(* Logix 5000 project; controller cal1615 1756-L62 rev 16.20; software revision 16.05; part 23 of 78 *)
(* tags used below, declared in another part *)
   FAULT : BOOL;   // Fault AFI
   HMI : BOOL;   // AFI HMI
   p01r09_pb_global_reset : BOOL;   // System Modes PB: Global Fault Reset
   p12_ai_exhaust_amps : REAL;   // Zone 2 Analog Input Exhaust Fan Amps
   p12_ai_exhaust_hz : REAL;   // Zone 2 Analog Input Exhaust Fan HZ
   p12_ai_exhaust_pct : REAL;   // Zone 2 Analog Input Exhaust Fan PCT
   p12_ai_exhaust_rpm : REAL;   // Zone 2 Analog Input Exhaust Fan RPM
   p12_ai_lfl : REAL;   // Zone 2 Analog Input Lower Flash Limit
   p12_ai_prs : REAL;   // Zone 2 Analog Input Pressure
   p12_ai_recirc_amps : REAL;   // Zone 2 Analog Input Recirc Fan Amps
   p12_ai_recirc_hz : REAL;   // Zone 2 Analog Input Supply Fan HZ
   p12_ai_recirc_pct : REAL;   // Zone 2 Analog Input Recirc Fan PCT
   p12_ai_recirc_rpm : REAL;   // Zone 2 Analog Input Recirc Fan RPM
   p12_ai_tc01 : REAL;   // Zone 2 Analog Input Control Thermocouple 1
   p12_ai_tc02 : REAL;   // Zone 2 Analog Input Control Thermocouple 2
   p12_ao_cv : REAL;   // Zone 2 Analog Output Control Valve
   p12_ao_exhaust_selected_speed : REAL;   // Zone 2 Analog Output Exhaust Fan VFD Selected Speed
   p12_ao_recirc_selected_speed : REAL;   // Zone 2 Analog Output Recirc Fan VFD Selected Speed
   p12_di_burner_auto : BOOL;   // Zone 2 Digital Input Burner Auto
   p12_di_exh : acs800_di_normal;   // Zone 2 Digital Inputs Exhaust Fan
   p12_di_recirc : acs800_di_normal;   // Zone 2 Digital Inputs Recirc Fan
   p12_dint_to_hmi : DINT[16];   // Zone 2 Temperature Control VFDs On
   p12_param_fast_to_soak : REAL;   // Zone 2 Parameter Fast to Soak Control
   p12_param_lfl_hhl : REAL;   // Zone 2 Parameter High High Lower Flash Limit
   p12_param_lfl_hl : REAL;   // Zone 2 Parameter High LFL Limit
   p12_param_pid1_ff : REAL;   // Zone 2 Parameter Fast PID Bias
   p12_param_pid1_kd : REAL;   // Zone 2 Parameter Fast PID Derivative Gain
   p12_param_pid1_ki : REAL;   // Zone 2 Parameter Fast PID Integral Gain
   p12_param_pid1_kp : REAL;   // Zone 2 Parameter Fast PID Proportional Gain
   p12_param_pid2_ff : REAL;   // Zone 2 Parameter Auto PID Bias
   p12_param_pid2_kd : REAL;   // Zone 2 Parameter Auto PID Derivative Gain
   p12_param_pid2_ki : REAL;   // Zone 2 Parameter Auto PID Integral Gain
   p12_param_pid2_kp : REAL;   // Zone 2 Parameter Auto PID Proportional Gain
   p12_param_shutdown_temp : REAL;   // Zone 2 Parameter Zone Shutdown Temperature
   p12_param_soak_to_fast : REAL;   // Zone 2 Parameter Soak to Fast Control
   p12_param_tc01_dev : REAL;   // Zone 2 Parameter Oven Temperature Deviation from Setpoint
   p12_param_tc01_hl : REAL;   // Zone 2 Parameter Process Air High Limit
   p12_param_tc01z : REAL;   // Zone 2 Parameter Process Temperature Zero Offset
   p12_param_tc02z : REAL;   // Zone 2 Parameter SupplyTemperature Zero Offset
   p12_param_zone_pressure : REAL;   // Zone 2 Parameter High Pressure LImit
   p12_real_to_hmi : REAL[112];   // Zone 2 Real to HMI
   p12r01 : routine;   // Zone 2 Main
   p12r05 : routine;   // Zone 2 Dint to HMI
   p12r05_exh_status : DINT;
   p12r05_recirc_status : DINT;
   p12r05_Temp_ctl_status : DINT;
   p12r05_timer_fault : TIMER[4];   // Zone 2 Dint to HMI Fault Delay
   p12r05_timer_warning : TIMER[4];   // Zone 2 Dint to HMI Warning Delay
   p12r06 : routine;   // Zone 2 Real to HMI
   p12r06_timer_fault : TIMER[4];   // Zone 2 Real to HMI Fault Delay
   p12r06_timer_warning : TIMER[4];   // Zone 2 Real to HMI Warning Delay
   p12r07 : routine;   // Zone 2 Alarms
   p12r07_timer_fault : TIMER[4];   // Zone 2 Alarms Fault Delay
   p12r07_timer_warning : TIMER[4];   // Zone 2 Alarms Warning Delay
   p12r20 : routine;   // Zone 2 Temp Sequence
   p12r20_state : DINT;   // Zone 2 Temperature Control State
   p12r20_status : DINT;   // Zone 2 Temperature Control Sequence Status
   p12r30 : routine;   // Zone 2 Temperature Control
   p12r30_cv_man_sp : REAL;   // Zone 2 Temperature Control Manual Heat Control Valve Setpoint
   p12r30_permissive_run : BOOL;   // Zone 2 Temperature Control Run Permissive
   p12r30_pid_temp : PID;   // Zone 2 Temperature Control PID
   p12r30_pid_temp_pv : REAL;   // Zone 2 Temperature Control PID Temp Process Variable
   p12r30_pid_temp_sp : REAL;   // Zone 2 Temperature Control PID Temperature Control Setpoint
   p12r30_request_heat : BOOL;   // Zone 2 Temperature Control Request Heat
   p12r31 : routine;   // Zone 2 Exhaust VFD
   p12r31_vfd_stopped : BOOL;   // Zone 2 Exhaust VFD VFD Stopped
   p12r32 : routine;   // Zone 2 Recirc VFD
   p12r32_vfd_stopped : BOOL;   // Zone 2 Recirc VFD VFD Stopped
(* P12_Zone_2, continued *)

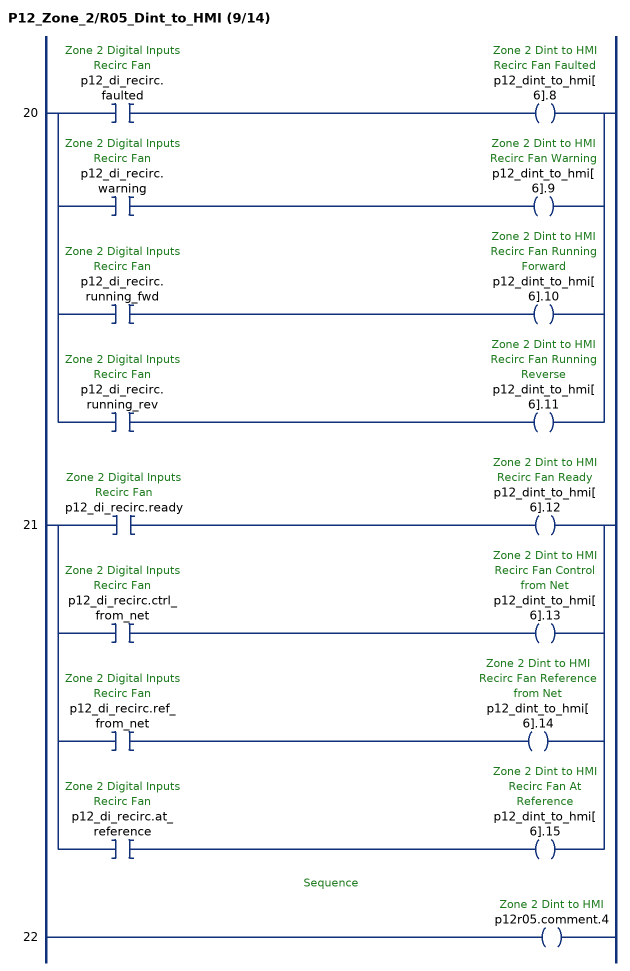
   [picture p388: P12_Zone_2/R05_Dint_to_HMI rungs 20-22]
   20: [XIC(p12_di_recirc.faulted) OTE(p12_dint_to_hmi[6].8) ,XIC(p12_di_recirc.warning) OTE(p12_dint_to_hmi[6].9) ,XIC(p12_di_recirc.running_fwd) OTE(p12_dint_to_hmi[6].10) ,XIC(p12_di_recirc.running_rev) OTE(p12_dint_to_hmi[6].11) ];
   21: [XIC(p12_di_recirc.ready) OTE(p12_dint_to_hmi[6].12) ,XIC(p12_di_recirc.ctrl_from_net) OTE(p12_dint_to_hmi[6].13) ,XIC(p12_di_recirc.ref_from_net) OTE(p12_dint_to_hmi[6].14) ,XIC(p12_di_recirc.at_reference) OTE(p12_dint_to_hmi[6].15) ];
   // Sequence
   22: OTE(p12r05.comment.4);
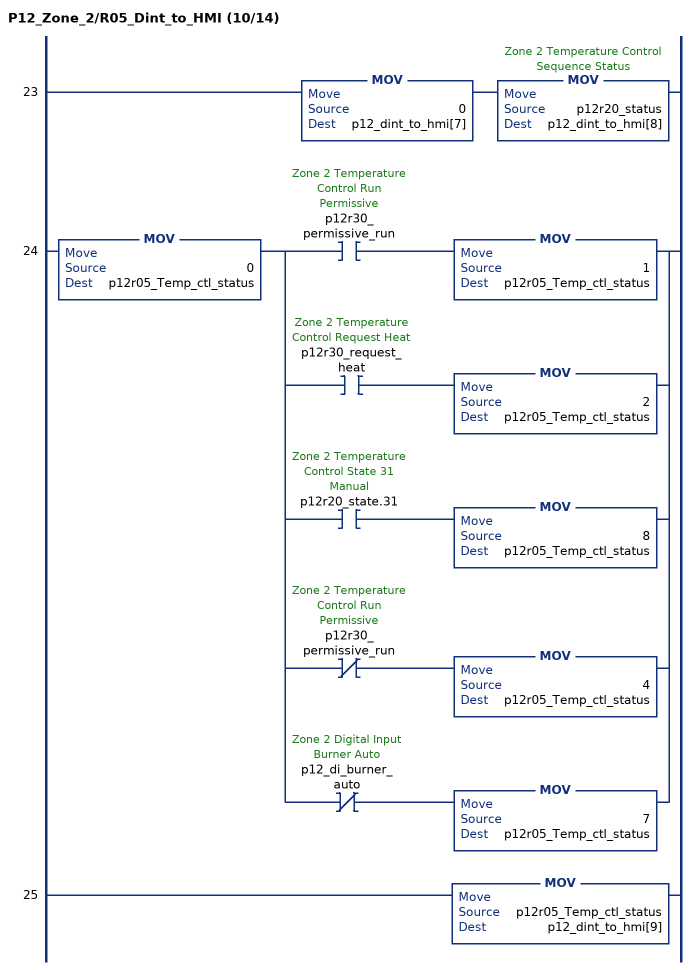
   23: MOV(0,p12_dint_to_hmi[7])MOV(p12r20_status,p12_dint_to_hmi[8]);
   24: MOV(0,p12r05_Temp_ctl_status)[XIC(p12r30_permissive_run) MOV(1,p12r05_Temp_ctl_status) ,XIC(p12r30_request_heat) MOV(2,p12r05_Temp_ctl_status) ,XIC(p12r20_state.31) MOV(8,p12r05_Temp_ctl_status) ,XIO(p12r30_permissive_run) MOV(4,p12r05_Temp_ctl_status) ,XIO(p12_di_burner_auto) MOV(7,p12r05_Temp_ctl_status) ];
   25: MOV(p12r05_Temp_ctl_status,p12_dint_to_hmi[9]);
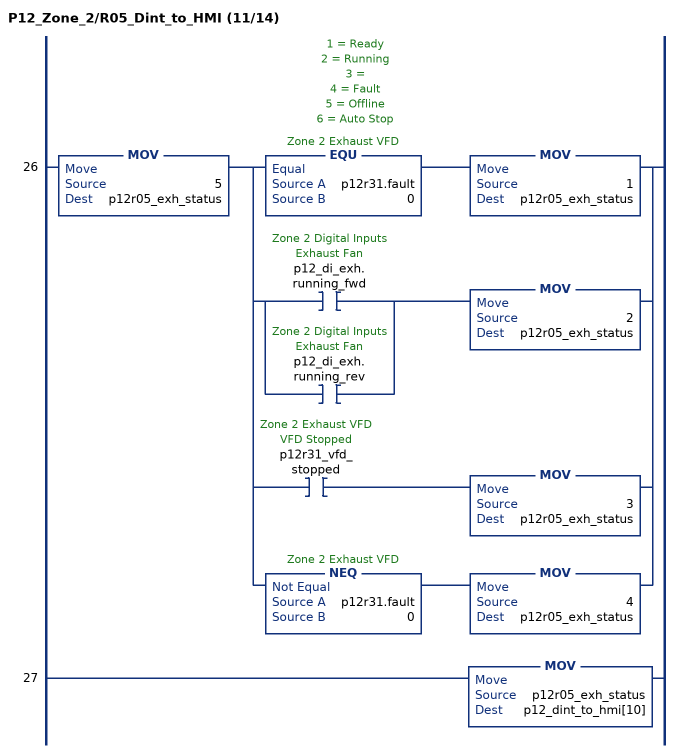
   // 1 = Ready
   // 2 = Running
   // 3 =
   // 4 = Fault
   // 5 = Offline
   // 6 = Auto Stop
   26: MOV(5,p12r05_exh_status)[EQU(p12r31.fault,0) MOV(1,p12r05_exh_status) ,[XIC(p12_di_exh.running_fwd) ,XIC(p12_di_exh.running_rev) ] MOV(2,p12r05_exh_status) ,XIC(p12r31_vfd_stopped) MOV(3,p12r05_exh_status) ,NEQ(p12r31.fault,0) MOV(4,p12r05_exh_status) ];
   27: MOV(p12r05_exh_status,p12_dint_to_hmi[10]);
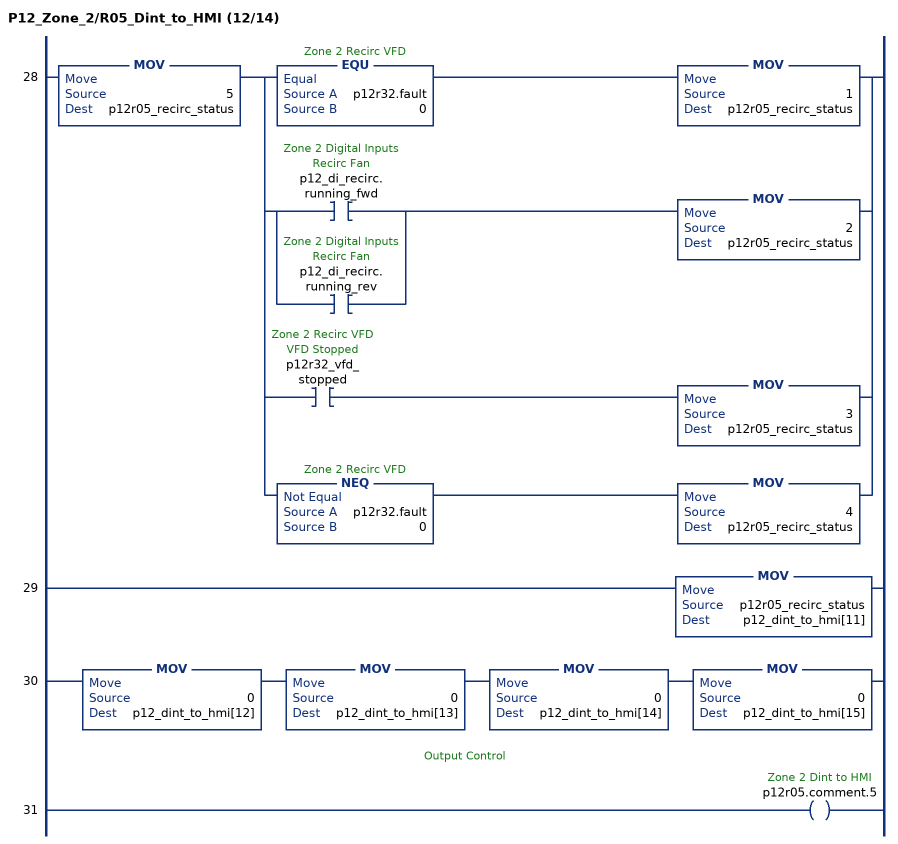
   28: MOV(5,p12r05_recirc_status)[EQU(p12r32.fault,0) MOV(1,p12r05_recirc_status) ,[XIC(p12_di_recirc.running_fwd) ,XIC(p12_di_recirc.running_rev) ] MOV(2,p12r05_recirc_status) ,XIC(p12r32_vfd_stopped) MOV(3,p12r05_recirc_status) ,NEQ(p12r32.fault,0) MOV(4,p12r05_recirc_status) ];
   29: MOV(p12r05_recirc_status,p12_dint_to_hmi[11]);
   30: MOV(0,p12_dint_to_hmi[12])MOV(0,p12_dint_to_hmi[13])MOV(0,p12_dint_to_hmi[14])MOV(0,p12_dint_to_hmi[15]);
   // Output Control
   31: OTE(p12r05.comment.5);
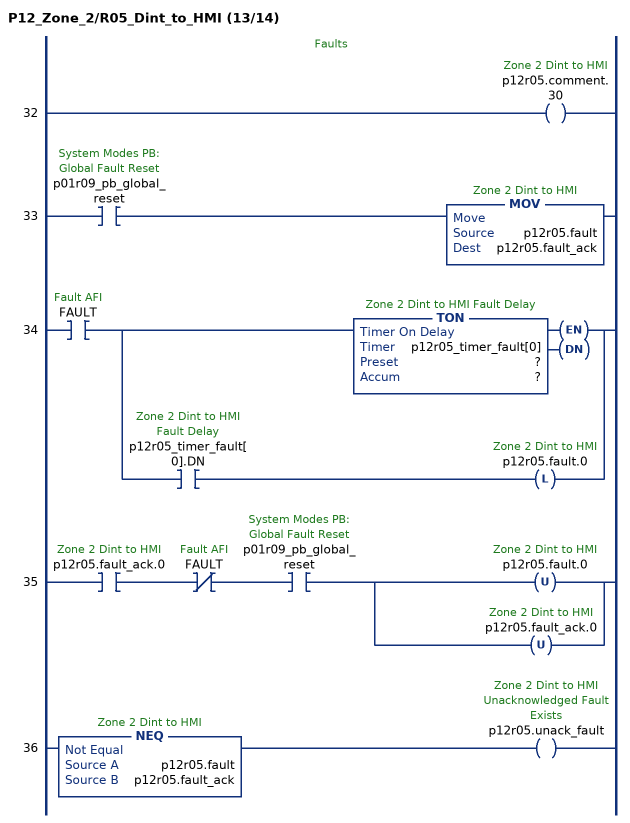
   // Faults
   32: OTE(p12r05.comment.30);
   33: XIC(p01r09_pb_global_reset)MOV(p12r05.fault,p12r05.fault_ack);
   34: XIC(FAULT)[TON(p12r05_timer_fault[0],?,?) ,XIC(p12r05_timer_fault[0].DN) OTL(p12r05.fault.0) ];
   35: XIC(p12r05.fault_ack.0)XIO(FAULT)XIC(p01r09_pb_global_reset)[OTU(p12r05.fault.0) ,OTU(p12r05.fault_ack.0) ];
   36: NEQ(p12r05.fault,p12r05.fault_ack)OTE(p12r05.unack_fault);
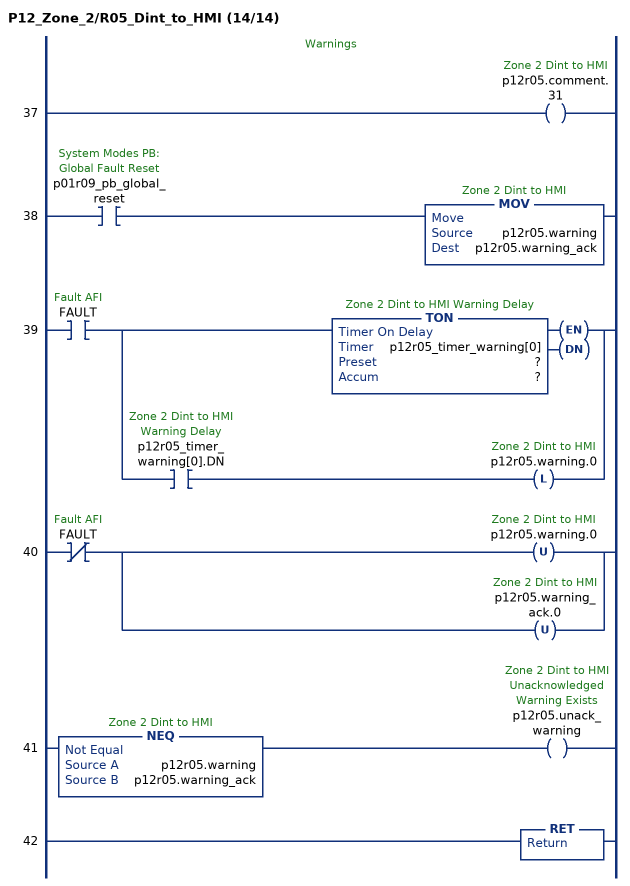
   // Warnings
   37: OTE(p12r05.comment.31);
   38: XIC(p01r09_pb_global_reset)MOV(p12r05.warning,p12r05.warning_ack);
   39: XIC(FAULT)[TON(p12r05_timer_warning[0],?,?) ,XIC(p12r05_timer_warning[0].DN) OTL(p12r05.warning.0) ];
   40: XIO(FAULT)[OTU(p12r05.warning.0) ,OTU(p12r05.warning_ack.0) ];
   41: NEQ(p12r05.warning,p12r05.warning_ack)OTE(p12r05.unack_warning);
   42: RET();
END_ROUTINE

ROUTINE R06_Real_to_HMI   (* ladder *)
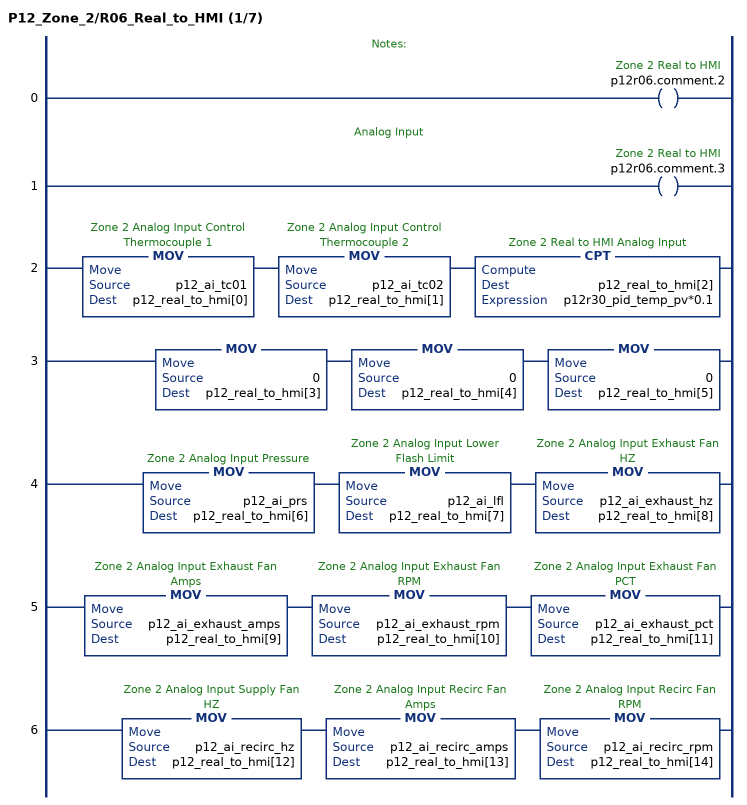
   // Notes:
   0: OTE(p12r06.comment.2);
   // Analog Input
   1: OTE(p12r06.comment.3);
   2: MOV(p12_ai_tc01,p12_real_to_hmi[0])MOV(p12_ai_tc02,p12_real_to_hmi[1])CPT(p12_real_to_hmi[2],p12r30_pid_temp_pv*0.1);
   3: MOV(0,p12_real_to_hmi[3])MOV(0,p12_real_to_hmi[4])MOV(0,p12_real_to_hmi[5]);
   4: MOV(p12_ai_prs,p12_real_to_hmi[6])MOV(p12_ai_lfl,p12_real_to_hmi[7])MOV(p12_ai_exhaust_hz,p12_real_to_hmi[8]);
   5: MOV(p12_ai_exhaust_amps,p12_real_to_hmi[9])MOV(p12_ai_exhaust_rpm,p12_real_to_hmi[10])MOV(p12_ai_exhaust_pct,p12_real_to_hmi[11]);
   6: MOV(p12_ai_recirc_hz,p12_real_to_hmi[12])MOV(p12_ai_recirc_amps,p12_real_to_hmi[13])MOV(p12_ai_recirc_rpm,p12_real_to_hmi[14]);
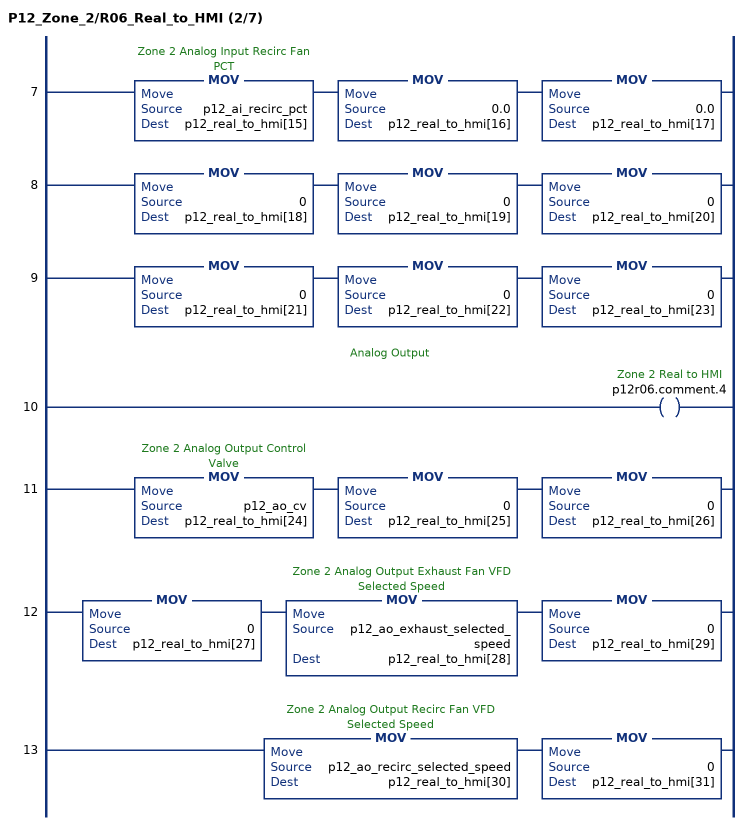
   7: MOV(p12_ai_recirc_pct,p12_real_to_hmi[15])MOV(0.0,p12_real_to_hmi[16])MOV(0.0,p12_real_to_hmi[17]);
   8: MOV(0,p12_real_to_hmi[18])MOV(0,p12_real_to_hmi[19])MOV(0,p12_real_to_hmi[20]);
   9: MOV(0,p12_real_to_hmi[21])MOV(0,p12_real_to_hmi[22])MOV(0,p12_real_to_hmi[23]);
   // Analog Output
   10: OTE(p12r06.comment.4);
   11: MOV(p12_ao_cv,p12_real_to_hmi[24])MOV(0,p12_real_to_hmi[25])MOV(0,p12_real_to_hmi[26]);
   12: MOV(0,p12_real_to_hmi[27])MOV(p12_ao_exhaust_selected_speed,p12_real_to_hmi[28])MOV(0,p12_real_to_hmi[29]);
   13: MOV(p12_ao_recirc_selected_speed,p12_real_to_hmi[30])MOV(0,p12_real_to_hmi[31]);
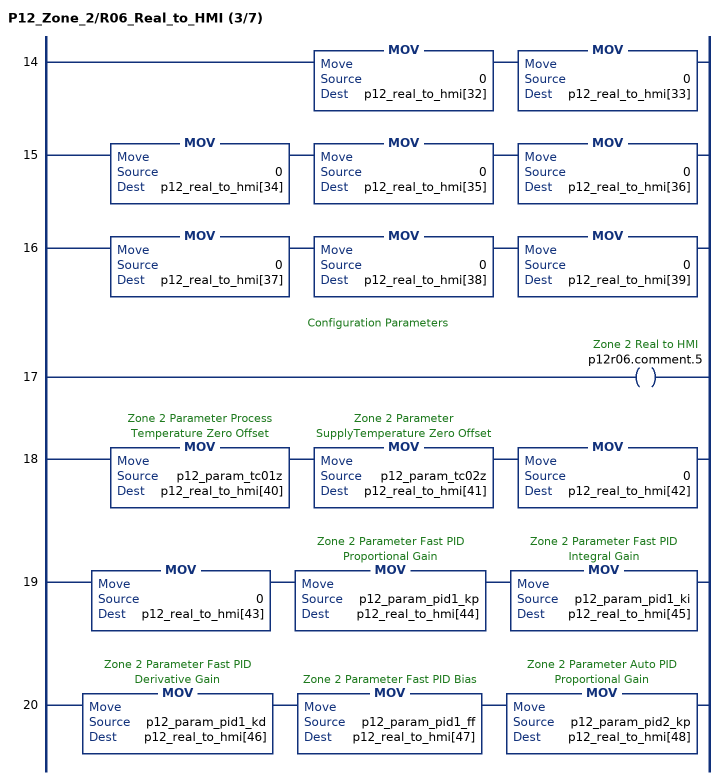
   14: MOV(0,p12_real_to_hmi[32])MOV(0,p12_real_to_hmi[33]);
   15: MOV(0,p12_real_to_hmi[34])MOV(0,p12_real_to_hmi[35])MOV(0,p12_real_to_hmi[36]);
   16: MOV(0,p12_real_to_hmi[37])MOV(0,p12_real_to_hmi[38])MOV(0,p12_real_to_hmi[39]);
   // Configuration Parameters
   17: OTE(p12r06.comment.5);
   18: MOV(p12_param_tc01z,p12_real_to_hmi[40])MOV(p12_param_tc02z,p12_real_to_hmi[41])MOV(0,p12_real_to_hmi[42]);
   19: MOV(0,p12_real_to_hmi[43])MOV(p12_param_pid1_kp,p12_real_to_hmi[44])MOV(p12_param_pid1_ki,p12_real_to_hmi[45]);
   20: MOV(p12_param_pid1_kd,p12_real_to_hmi[46])MOV(p12_param_pid1_ff,p12_real_to_hmi[47])MOV(p12_param_pid2_kp,p12_real_to_hmi[48]);
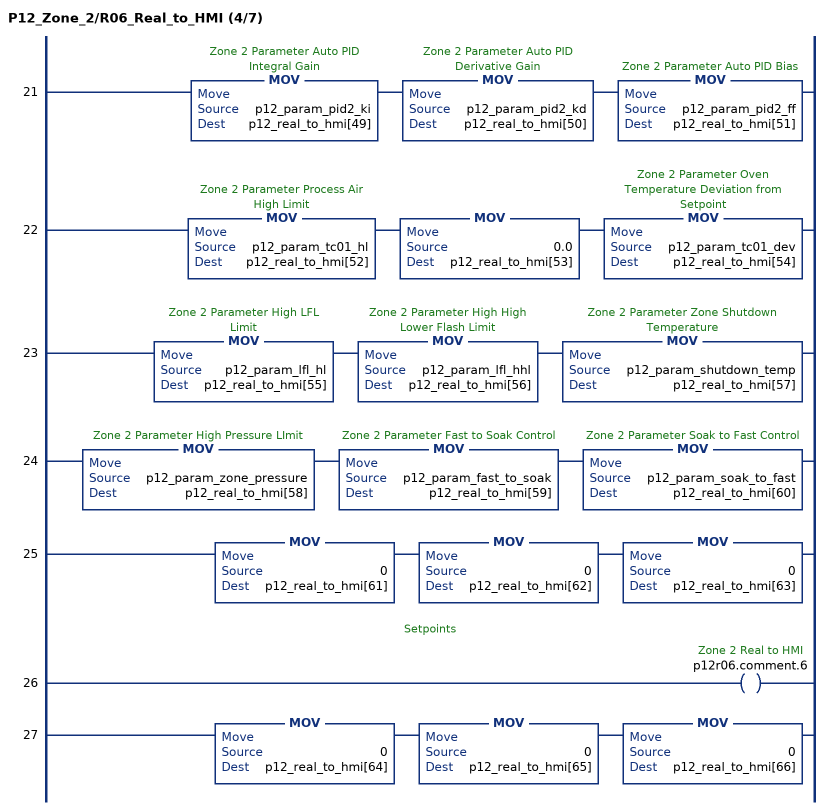
   21: MOV(p12_param_pid2_ki,p12_real_to_hmi[49])MOV(p12_param_pid2_kd,p12_real_to_hmi[50])MOV(p12_param_pid2_ff,p12_real_to_hmi[51]);
   22: MOV(p12_param_tc01_hl,p12_real_to_hmi[52])MOV(0.0,p12_real_to_hmi[53])MOV(p12_param_tc01_dev,p12_real_to_hmi[54]);
   23: MOV(p12_param_lfl_hl,p12_real_to_hmi[55])MOV(p12_param_lfl_hhl,p12_real_to_hmi[56])MOV(p12_param_shutdown_temp,p12_real_to_hmi[57]);
   24: MOV(p12_param_zone_pressure,p12_real_to_hmi[58])MOV(p12_param_fast_to_soak,p12_real_to_hmi[59])MOV(p12_param_soak_to_fast,p12_real_to_hmi[60]);
   25: MOV(0,p12_real_to_hmi[61])MOV(0,p12_real_to_hmi[62])MOV(0,p12_real_to_hmi[63]);
   // Setpoints
   26: OTE(p12r06.comment.6);
   27: MOV(0,p12_real_to_hmi[64])MOV(0,p12_real_to_hmi[65])MOV(0,p12_real_to_hmi[66]);
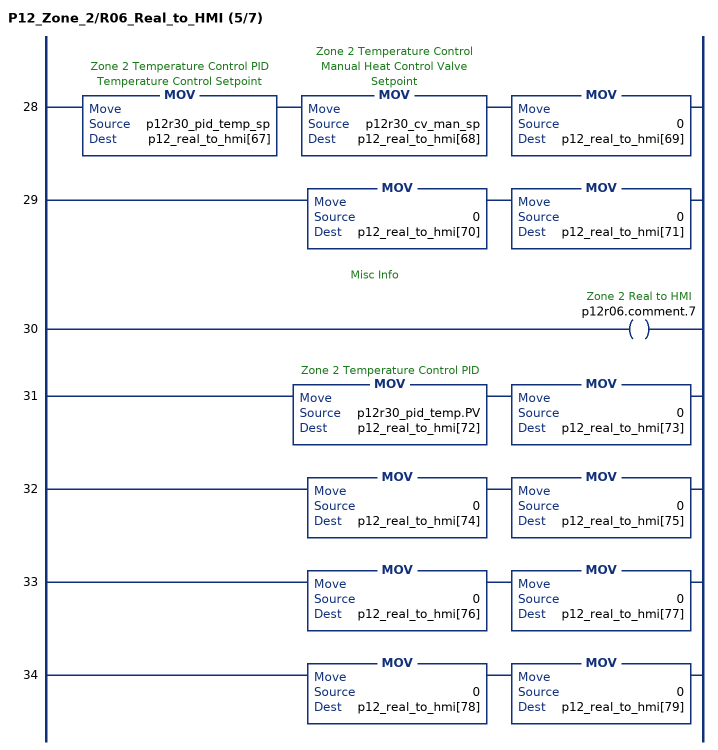
   28: MOV(p12r30_pid_temp_sp,p12_real_to_hmi[67])MOV(p12r30_cv_man_sp,p12_real_to_hmi[68])MOV(0,p12_real_to_hmi[69]);
   29: MOV(0,p12_real_to_hmi[70])MOV(0,p12_real_to_hmi[71]);
   // Misc Info
   30: OTE(p12r06.comment.7);
   31: MOV(p12r30_pid_temp.PV,p12_real_to_hmi[72])MOV(0,p12_real_to_hmi[73]);
   32: MOV(0,p12_real_to_hmi[74])MOV(0,p12_real_to_hmi[75]);
   33: MOV(0,p12_real_to_hmi[76])MOV(0,p12_real_to_hmi[77]);
   34: MOV(0,p12_real_to_hmi[78])MOV(0,p12_real_to_hmi[79]);
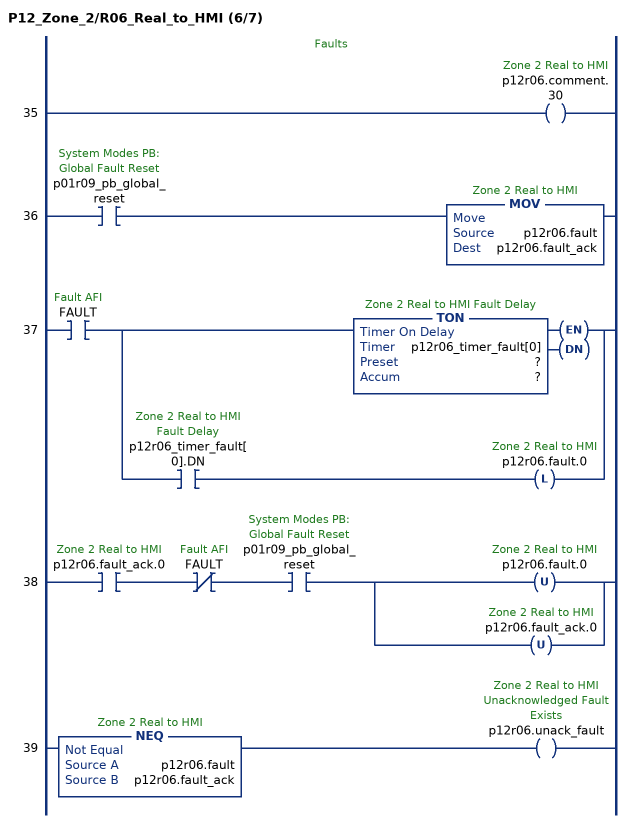
   // Faults
   35: OTE(p12r06.comment.30);
   36: XIC(p01r09_pb_global_reset)MOV(p12r06.fault,p12r06.fault_ack);
   37: XIC(FAULT)[TON(p12r06_timer_fault[0],?,?) ,XIC(p12r06_timer_fault[0].DN) OTL(p12r06.fault.0) ];
   38: XIC(p12r06.fault_ack.0)XIO(FAULT)XIC(p01r09_pb_global_reset)[OTU(p12r06.fault.0) ,OTU(p12r06.fault_ack.0) ];
   39: NEQ(p12r06.fault,p12r06.fault_ack)OTE(p12r06.unack_fault);
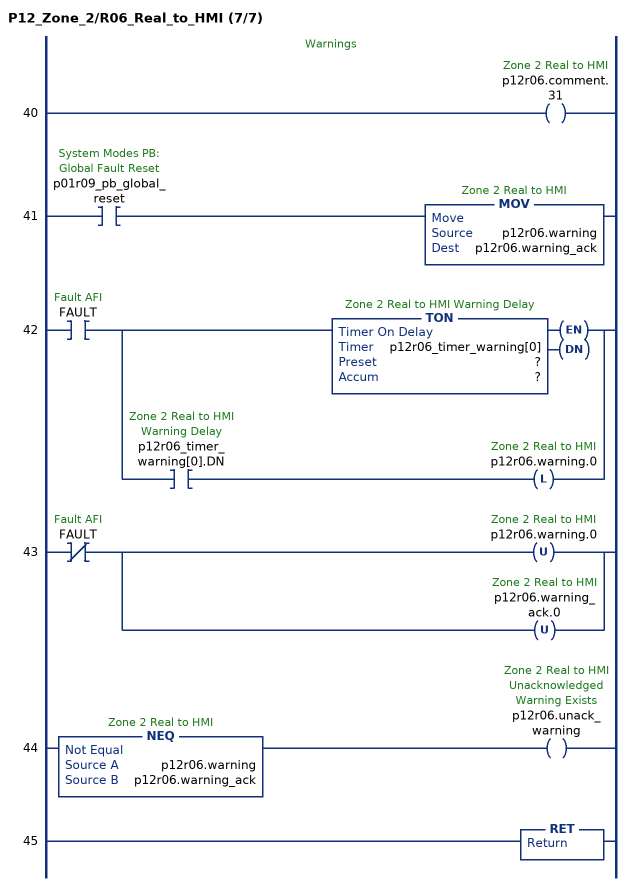
   // Warnings
   40: OTE(p12r06.comment.31);
   41: XIC(p01r09_pb_global_reset)MOV(p12r06.warning,p12r06.warning_ack);
   42: XIC(FAULT)[TON(p12r06_timer_warning[0],?,?) ,XIC(p12r06_timer_warning[0].DN) OTL(p12r06.warning.0) ];
   43: XIO(FAULT)[OTU(p12r06.warning.0) ,OTU(p12r06.warning_ack.0) ];
   44: NEQ(p12r06.warning,p12r06.warning_ack)OTE(p12r06.unack_warning);
   45: RET();
END_ROUTINE

ROUTINE R07_Alarms   (* ladder *)
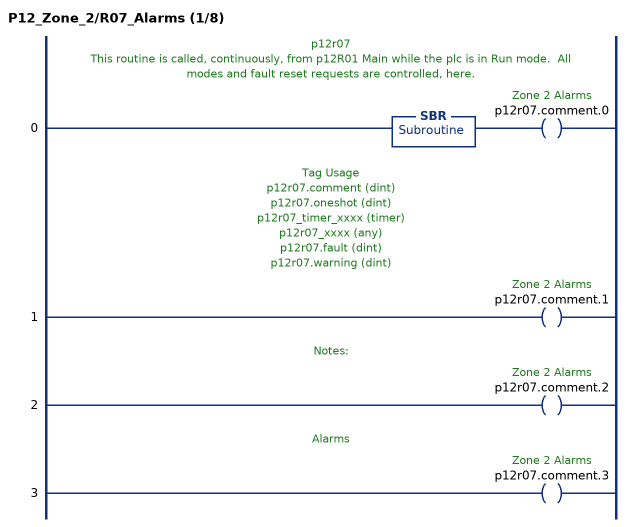
   // p12r07
   // This routine is called, continuously, from p12R01 Main while the plc is in Run mode.  All modes and fault reset requests are controlled, here.
   0: SBR()OTE(p12r07.comment.0);
   // Tag Usage
   // p12r07.comment (dint)
   // p12r07.oneshot (dint)
   // p12r07_timer_xxxx (timer)
   // p12r07_xxxx (any)
   // p12r07.fault (dint)
   // p12r07.warning (dint)
   1: OTE(p12r07.comment.1);
   // Notes:
   2: OTE(p12r07.comment.2);
   // Alarms
   3: OTE(p12r07.comment.3);
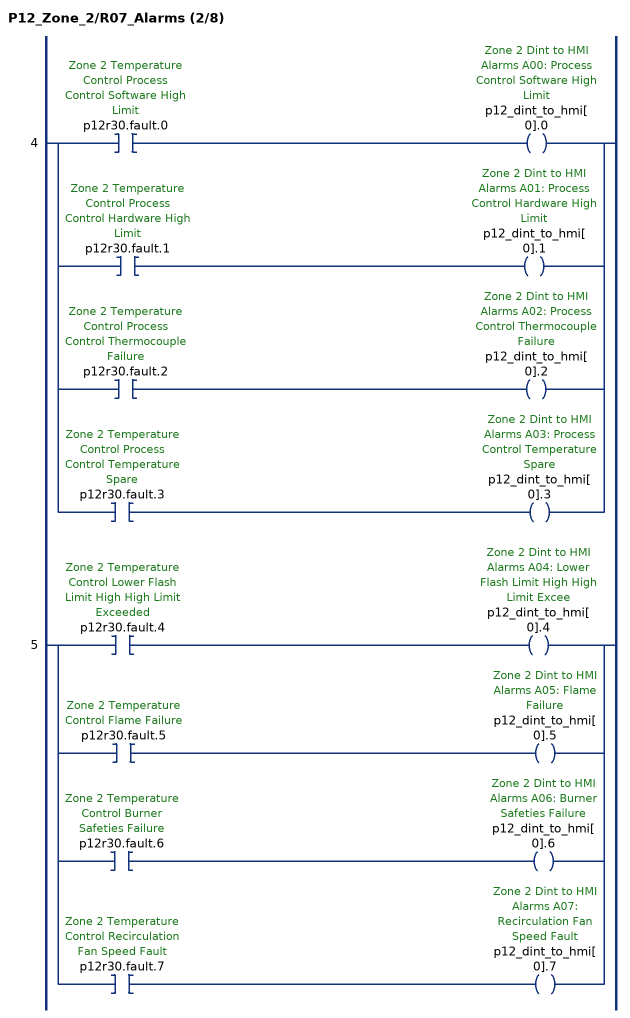
   4: [XIC(p12r30.fault.0) OTE(p12_dint_to_hmi[0].0) ,XIC(p12r30.fault.1) OTE(p12_dint_to_hmi[0].1) ,XIC(p12r30.fault.2) OTE(p12_dint_to_hmi[0].2) ,XIC(p12r30.fault.3) OTE(p12_dint_to_hmi[0].3) ];
   5: [XIC(p12r30.fault.4) OTE(p12_dint_to_hmi[0].4) ,XIC(p12r30.fault.5) OTE(p12_dint_to_hmi[0].5) ,XIC(p12r30.fault.6) OTE(p12_dint_to_hmi[0].6) ,XIC(p12r30.fault.7) OTE(p12_dint_to_hmi[0].7) ];
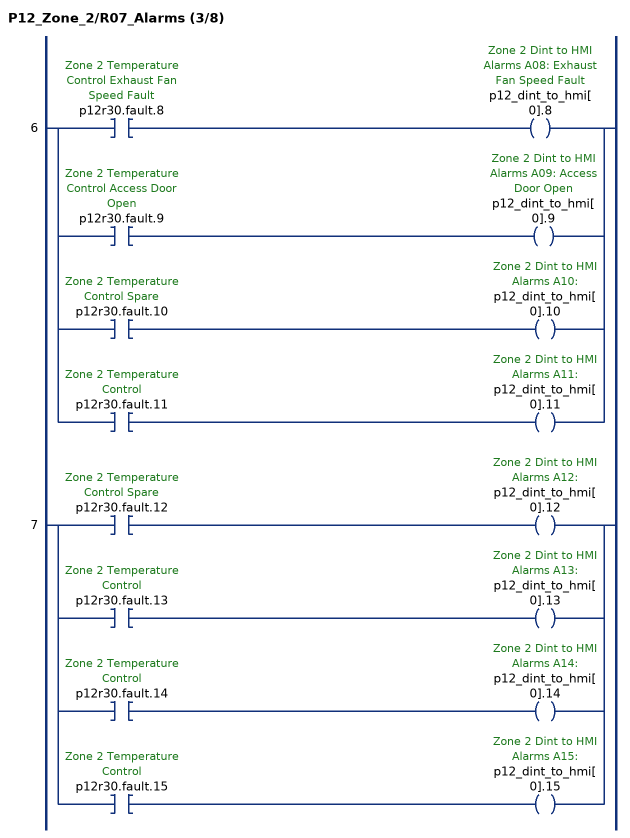
   6: [XIC(p12r30.fault.8) OTE(p12_dint_to_hmi[0].8) ,XIC(p12r30.fault.9) OTE(p12_dint_to_hmi[0].9) ,XIC(p12r30.fault.10) OTE(p12_dint_to_hmi[0].10) ,XIC(p12r30.fault.11) OTE(p12_dint_to_hmi[0].11) ];
   7: [XIC(p12r30.fault.12) OTE(p12_dint_to_hmi[0].12) ,XIC(p12r30.fault.13) OTE(p12_dint_to_hmi[0].13) ,XIC(p12r30.fault.14) OTE(p12_dint_to_hmi[0].14) ,XIC(p12r30.fault.15) OTE(p12_dint_to_hmi[0].15) ];
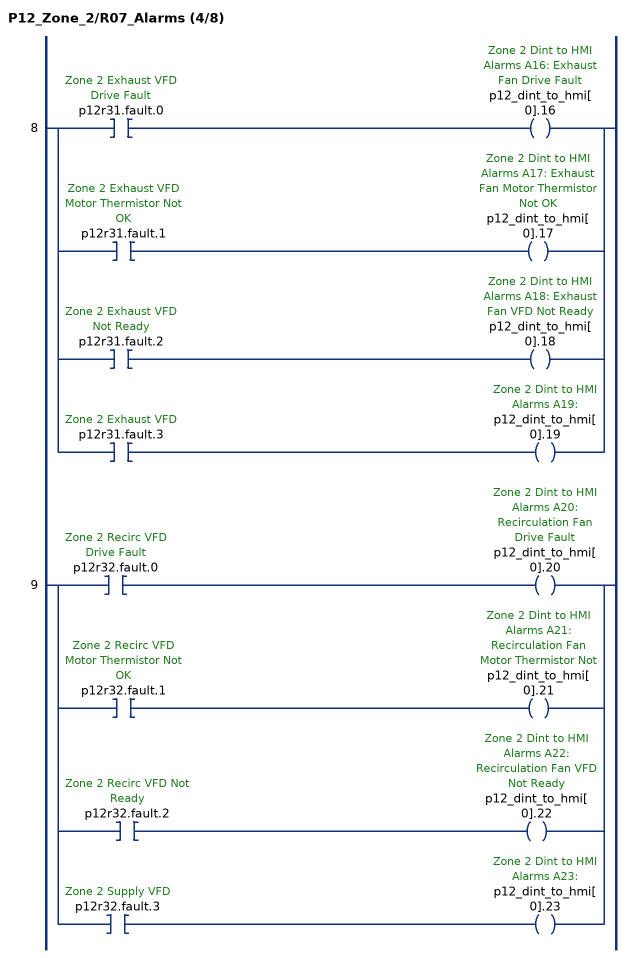
   8: [XIC(p12r31.fault.0) OTE(p12_dint_to_hmi[0].16) ,XIC(p12r31.fault.1) OTE(p12_dint_to_hmi[0].17) ,XIC(p12r31.fault.2) OTE(p12_dint_to_hmi[0].18) ,XIC(p12r31.fault.3) OTE(p12_dint_to_hmi[0].19) ];
   9: [XIC(p12r32.fault.0) OTE(p12_dint_to_hmi[0].20) ,XIC(p12r32.fault.1) OTE(p12_dint_to_hmi[0].21) ,XIC(p12r32.fault.2) OTE(p12_dint_to_hmi[0].22) ,XIC(p12r32.fault.3) OTE(p12_dint_to_hmi[0].23) ];
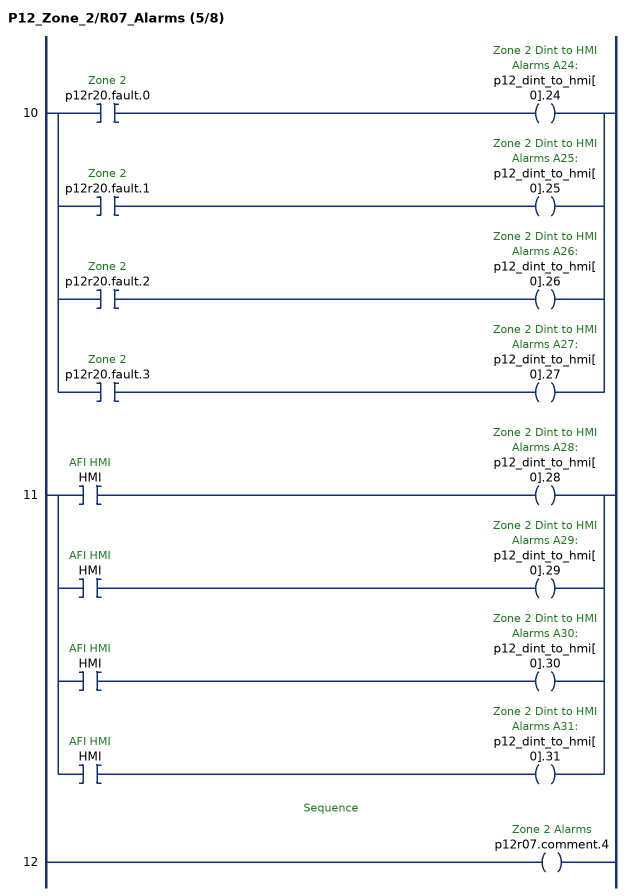
   10: [XIC(p12r20.fault.0) OTE(p12_dint_to_hmi[0].24) ,XIC(p12r20.fault.1) OTE(p12_dint_to_hmi[0].25) ,XIC(p12r20.fault.2) OTE(p12_dint_to_hmi[0].26) ,XIC(p12r20.fault.3) OTE(p12_dint_to_hmi[0].27) ];
   11: [XIC(HMI) OTE(p12_dint_to_hmi[0].28) ,XIC(HMI) OTE(p12_dint_to_hmi[0].29) ,XIC(HMI) OTE(p12_dint_to_hmi[0].30) ,XIC(HMI) OTE(p12_dint_to_hmi[0].31) ];
   // Sequence
   12: OTE(p12r07.comment.4);
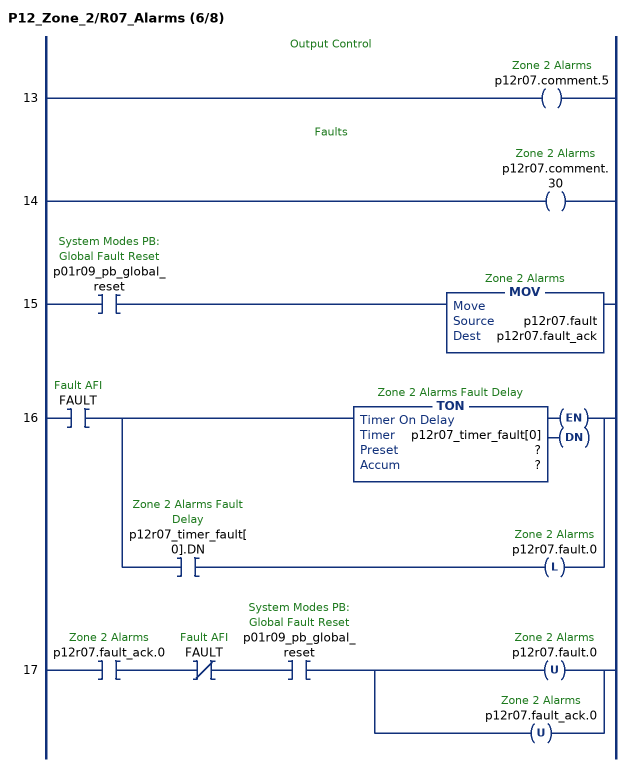
   // Output Control
   13: OTE(p12r07.comment.5);
   // Faults
   14: OTE(p12r07.comment.30);
   15: XIC(p01r09_pb_global_reset)MOV(p12r07.fault,p12r07.fault_ack);
   16: XIC(FAULT)[TON(p12r07_timer_fault[0],?,?) ,XIC(p12r07_timer_fault[0].DN) OTL(p12r07.fault.0) ];
   17: XIC(p12r07.fault_ack.0)XIO(FAULT)XIC(p01r09_pb_global_reset)[OTU(p12r07.fault.0) ,OTU(p12r07.fault_ack.0) ];
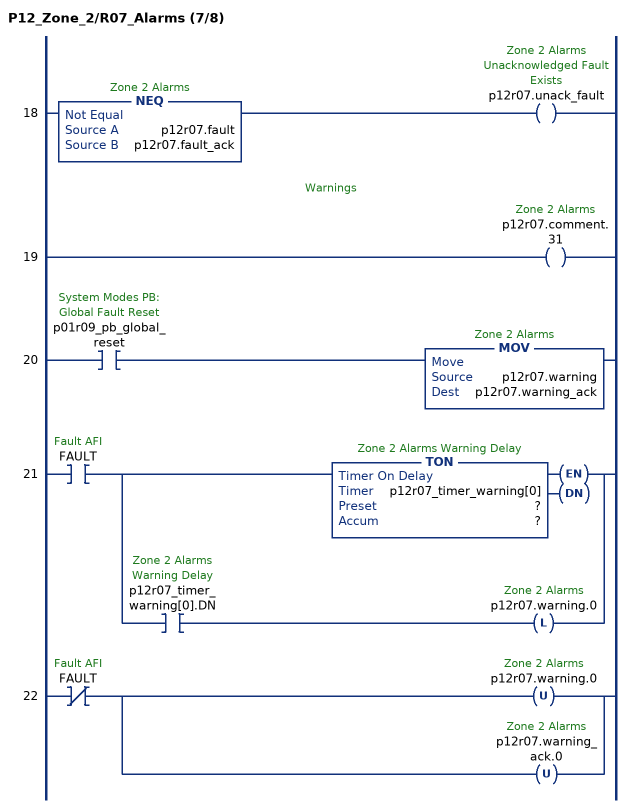
   18: NEQ(p12r07.fault,p12r07.fault_ack)OTE(p12r07.unack_fault);
   // Warnings
   19: OTE(p12r07.comment.31);
   20: XIC(p01r09_pb_global_reset)MOV(p12r07.warning,p12r07.warning_ack);
   21: XIC(FAULT)[TON(p12r07_timer_warning[0],?,?) ,XIC(p12r07_timer_warning[0].DN) OTL(p12r07.warning.0) ];
   22: XIO(FAULT)[OTU(p12r07.warning.0) ,OTU(p12r07.warning_ack.0) ];
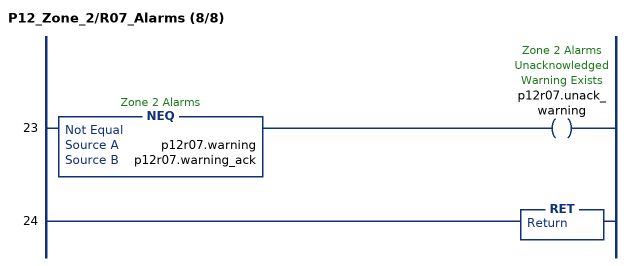
   23: NEQ(p12r07.warning,p12r07.warning_ack)OTE(p12r07.unack_warning);
   24: RET();
END_ROUTINE
